FUNCTION_BLOCK OPCUA_READ_1322467A4CC663E9C (* Generic Interface Function Block Type *)
  (* Standard: 61499-2 *)
  (* Version 0.0, 31/08/2020, Administrator, nxtControl GmbH, Template *)
  PACKAGE Main;
  (* Compiler Cpp nxtControl builtin 1.0 *)
  {SET_ATTRIBUTE(Runtime.FBType.ImplementingType, Standard.OPCUAClient#DYNGEN_OPCUA_READ)}
  {SET_ATTRIBUTE(Configuration.GenericFBType.InterfaceParams, Standard.OPCUAClient#CNTX:=2;VALUE${CNTX$}:BOOL,BOOL)}
  {SET_ATTRIBUTE(Configuration.FBType.IsKind.OPCUA_CLIENT, )}
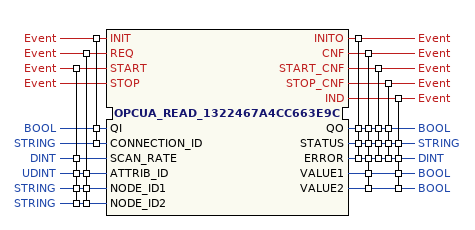
  EVENT_INPUT
    INIT WITH QI, CONNECTION_ID; (* Triggers initialization or deinitialization of FB *)
    REQ WITH ATTRIB_ID, NODE_ID1, NODE_ID2; (* Triggers acyclic reading *)
    START WITH SCAN_RATE, ATTRIB_ID, NODE_ID1, NODE_ID2; (* riggers cyclic reading (polling) *)
    STOP; (* Stops cyclic reading *)
  END_EVENT
  EVENT_OUTPUT
    INITO WITH QO, STATUS, ERROR; (* Confirmation of initialization or deinitialization of FB *)
    CNF WITH QO, STATUS, ERROR, VALUE1, VALUE2; (* Confirmation of completion of acyclic read operation *)
    START_CNF WITH QO, STATUS, ERROR; (* Triggered whenever a cyclic read operation is initiated *)
    STOP_CNF WITH QO, STATUS, ERROR; (* Triggered whenever a cyclic read operation is stopped *)
    IND WITH VALUE1, VALUE2, ERROR, STATUS; (* Indication event for cyclic read operation *)
  END_EVENT
  VAR_INPUT
    QI : BOOL; (* Qualifier Input *)
    CONNECTION_ID : STRING; (* Connection  ID associated with server to be accessed *)
    SCAN_RATE : DINT; (* Scanning/polling rate in milliseconds of cyclic read operation *)
    ATTRIB_ID : UDINT; (* Node attribute* ID to be read (13 i.e. node value attribute if not specified) *) {SET_ATTRIBUTE(Configuration.Parameter.DefaultConstant, 13)}
    NODE_ID1 : STRING; (* Node address of node to be accessed (see Node Addressing section for details) *)
    NODE_ID2 : STRING; (* Node address of node to be accessed (see Node Addressing section for details) *)
  END_VAR
  VAR_OUTPUT
    QO : BOOL; (* Output event qualifier *)
    STATUS : STRING; (* Displays status of FB *)
    ERROR : DINT; (* Displays error code for last performed read operation. See section FB Error Codes for description of error codes *)
    VALUE1 : BOOL; (* Value of the node attribute read during the last successful read operation *)
    VALUE2 : BOOL; (* Value of the node attribute read during the last successful read operation *)
  END_VAR
  EC_STATES
    START;
  END_STATES
END_FUNCTION_BLOCK
